KUKA KRL data list: Help.dat

&ACCESS RVO
&REL 1
&PARAM EDITMASK = *
&PARAM TEMPLATE = C:\KRC\Roboter\Template\vorgabe

DEFDAT Help
;FOLD EXTERNAL DECLARATIONS;%{PE}%MKUKATPBASIS,%CEXT,%VCOMMON,%P
;START AUTOGENERATED -- DO NOT CHANGE -- Gripper-&SpotTech vorgabe Vorgabe_dat_Grp&Spot.add InsertGripperTechGlobals
;FOLD GRIPPERTECH EXT
EXT  H50 (INT  :IN,INT  :IN,INT  :IN,GRP_TYP  :IN )
;ENDFOLD (GRIPPERTECH EXT)
;END AUTOGENERATED -- DO NOT CHANGE -- (Gripper-&SpotTech vorgabe Vorgabe_dat_Grp&Spot.add InsertGripperTechGlobals)
;START AUTOGENERATED -- DO NOT CHANGE -- Gripper-&SpotTech vorgabe Vorgabe_dat_Grp&Spot.add InsertSpotTechGlobals
;FOLD SPOTTECH EXT
EXT  USERSPOT (S_COMMAND  :IN,SPOT_TYPE  :IN )
;ENDFOLD (SPOTTECH EXT)
;END AUTOGENERATED -- DO NOT CHANGE -- (Gripper-&SpotTech vorgabe Vorgabe_dat_Grp&Spot.add InsertSpotTechGlobals)
;FOLD BASISTECH EXT;%{PE}%MKUKATPBASIS,%CEXT,%VEXT,%P
EXT  BAS (BAS_COMMAND  :IN,REAL  :IN )
DECL INT SUCCESS
;ENDFOLD (BASISTECH EXT)
;FOLD USER EXT;%{E}%MKUKATPUSER,%CEXT,%VEXT,%P
;Make your modifications here;ENDFOLD (USER EXT)
;ENDFOLD (EXTERNAL DECLARATIONS)

DECL BASIS_SUGG_T LAST_BASIS={POINT1[] "P2                      ",POINT2[] "P2                      ",CP_PARAMS[] "CPDAT0                  ",PTP_PARAMS[] "PDAT2                   ",CONT[] "C_DIS                   ",CP_VEL[] "2.0                     ",PTP_VEL[] "10                      ",SYNC_PARAMS[] "SYNCDAT                 ",SPL_NAME[] "S0                      ",A_PARAMS[] "ADAT0                   "}
